FUNCTION TryConvert_UDINT_TO_LINT : BOOL
VAR_INPUT
	in : UDINT;
	out : REFERENCE TO LINT;
END_VAR

out := UDINT_TO_LINT(in);
TryConvert_UDINT_TO_LINT := TRUE;

END_FUNCTION

(* stored: Version 1.1.0.1, ProductVersion 3.1.4024.12
   POU TryConvert_UDINT_TO_LINT: Id {0746cc98-4efc-4466-93ae-7606a62a5e52}, SpecialFunc None *)
